// TIA Portal V17 export
BLOCK "FC_NativeScl"   // ObjectSW18, SCL
// native SCL body passthrough
BEGIN
END_BLOCK
